% RSLogix 500 project Fail Safe.RSS, saved by version 10.00.00.00 %
PROJECT "UNTITLED"    % processor: Bul.1763 MicroLogix 1100 Series B %

PROGRAM FILES
  LAD 2 "INVERTS"  4 rungs
  LAD 3 "SIM"  2 rungs
  LAD 4 "ERR"  7 rungs  % Simulation %
  LAD 5 "MAIN"  2 rungs

DATA FILES
  O0 OUTPUT  4 elements
  I1 INPUT  6 elements
  S2 STATUS  66 elements
  B3 BINARY  11 elements
  T4 TIMER  17 elements
  C5 COUNTER  11 elements
  R6 CONTROL  1 elements
  N7 INTEGER  11 elements
  F8 FLOAT  1 elements

LADDER 2 "INVERTS"
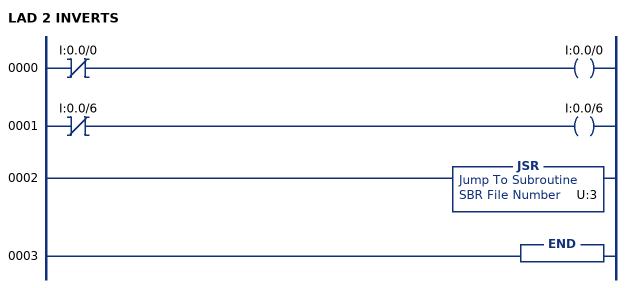
% Rung: 0 %
SOR XIO I:0.0/0 OTE I:0.0/0 EOR
% Rung: 1 %
SOR XIO I:0.0/6 OTE I:0.0/6 EOR
% Rung: 2 %
SOR JSR U:3 EOR
% Rung: 3 %
SOR END EOR

LADDER 3 "SIM"
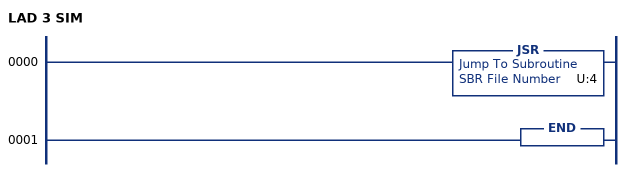
% Rung: 0 %
SOR JSR U:4 EOR
% Rung: 1 %
SOR END EOR

LADDER 4 "ERR"    % Simulation %
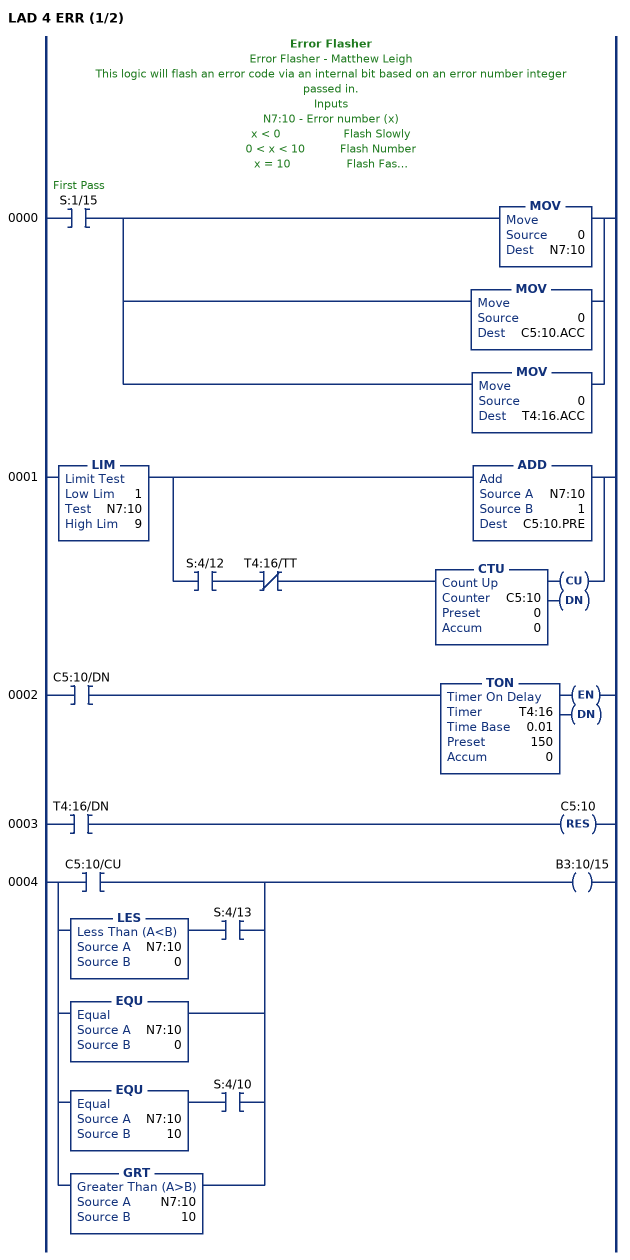
% Rung: 0 %
% TITLE: Error Flasher %
% Error Flasher - Matthew Leigh
% This logic will flash an error code via an internal bit based on an error number integer passed in.
% 
% Inputs
%    N7:10 - Error number (x)
%       x < 0                  Flash Slowly
%       0 < x < 10          Flash Number
%       x = 10                Flash Fast
%       x = 0 or x > 10   On Solid
% 
% Outputs
%    B3:10/15 - Flashing bit %
SOR XIC S:1/15 BST MOV 0 N7:10 NXB MOV 0 C5:10.ACC NXB MOV 0 T4:16.ACC BND EOR
%   S:1/15  "First Pass" %
% Rung: 1 %
SOR LIM 1 N7:10 9 BST ADD N7:10 1 C5:10.PRE NXB XIC S:4/12 XIO T4:16/TT CTU C5:10 0 0 BND EOR
% Rung: 2 %
SOR XIC C5:10/DN TON T4:16 0.01 150 0 EOR
% Rung: 3 %
SOR XIC T4:16/DN RES C5:10 EOR
% Rung: 4 %
SOR BST XIC C5:10/CU NXB LES N7:10 0 XIC S:4/13 NXB EQU N7:10 0 NXB EQU N7:10 10 XIC S:4/10 NXB GRT N7:10 10 BND OTE B3:10/15 EOR

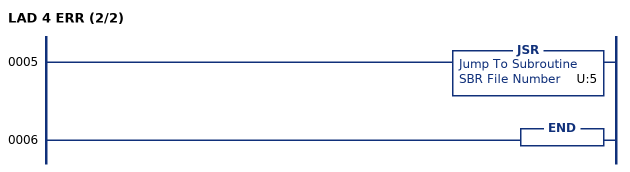
% Rung: 5 %
SOR JSR U:5 EOR
% Rung: 6 %
SOR END EOR

LADDER 5 "MAIN"
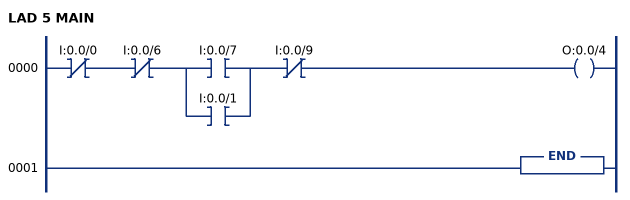
% Rung: 0 %
SOR XIO I:0.0/0 XIO I:0.0/6 BST XIC I:0.0/7 NXB XIC I:0.0/1 BND XIO I:0.0/9 OTE O:0.0/4 EOR
% Rung: 1 %
SOR END EOR

DATA TABLE (non-zero values as saved)
DATA T4
% .PRE .ACC %
% T4:16 % 150 0
